PROGRAM P_HMI_Polling
VAR

END_VAR


Global_variables.HMI_Servo1_Pos := io.DriveAxis1.NcToPlc.ActPos;
Global_variables.HMI_Servo1_Vel := io.DriveAxis1.NcToPlc.ActVelo;
Global_variables.HMI_Servo1_Torque := io.DriveAxis1.NcToPlc.ActTorque;

Global_variables.HMI_Servo2_Pos := io.DriveAxis2.NcToPlc.ActPos;
Global_variables.HMI_Servo2_Vel := io.DriveAxis1.NcToPlc.ActVelo;
Global_variables.HMI_Servo2_Torque := io.DriveAxis2.NcToPlc.ActTorque;

io.PowerEnabled := Global_variables.HmiButtonData0.2; 
Control.b_EnableServosReq := Global_variables.HmiButtonData0.2;
Control.b_RequestServoReset := Global_variables.HmiButtonData0.3;
IO.Laser_mm := UINT_TO_LREAL(io.LaserDistanceValue)  / 10.0;


Global_variables.HmiBoolDword0.0 := io.DriveEnabled1;
Global_variables.HmiBoolDword0.1 := io.DriveFaulted1;
Global_variables.HmiBoolDword0.2 := io.DriveEnabled2;
Global_variables.HmiBoolDword0.3 := io.DriveFaulted2;
Global_variables.HmiBoolDword0.4 := Global_variables.b_GearIn;
Global_variables.HmiBoolDword0.5 := control.b_Servos_Halted;
Global_variables.HmiBoolDword0.6 := control.b_EnableServosFinal;
Global_variables.HmiBoolDword0.7 := p_Faultmonitoring.b_Faulted;

END_PROGRAM

(* stored: Version 1.1.0.1, ProductVersion 3.1.4024.4
   POU P_HMI_Polling: Id {6c3f4490-3ab2-422f-af2f-6459f65a48e9}, SpecialFunc None *)
